FUNCTION_BLOCK Model (* Composite Function Block Type *)
  (* Standard: 61499-2 *)
  (* Version 0.0, 6/17/2016, Andrei, nxtControl GmbH, template *)
  PACKAGE Main;
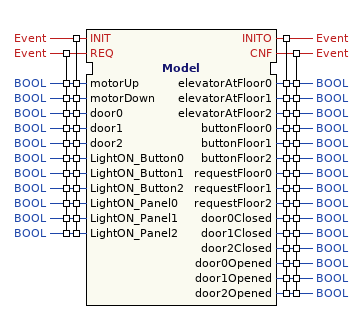
  EVENT_INPUT
    INIT WITH motorUp, motorDown, door0, door1, door2, LightON_Button0, LightON_Button1, LightON_Button2, LightON_Panel0, LightON_Panel1, LightON_Panel2; (* Initialization Request *)
    REQ WITH motorUp, motorDown, door0, door1, door2, LightON_Button0, LightON_Button1, LightON_Button2, LightON_Panel0, LightON_Panel1, LightON_Panel2; (* Normal Execution Request *)
  END_EVENT
  EVENT_OUTPUT
    INITO WITH buttonFloor0, buttonFloor1, buttonFloor2, requestFloor0, requestFloor1, requestFloor2, elevatorAtFloor0, elevatorAtFloor1, elevatorAtFloor2, door0Closed, door1Closed, door2Closed, door0Opened, door1Opened, door2Opened; (* Initialization Confirm *)
    CNF WITH buttonFloor0, buttonFloor1, buttonFloor2, requestFloor0, requestFloor1, requestFloor2, elevatorAtFloor0, elevatorAtFloor1, elevatorAtFloor2, door0Closed, door1Closed, door2Closed, door0Opened, door1Opened, door2Opened; (* Execution Confirmation *)
  END_EVENT
  VAR_INPUT
    motorUp : BOOL; (* Input event qualifier *)
    motorDown : BOOL;
    door0 : BOOL;
    door1 : BOOL;
    door2 : BOOL;
    LightON_Button0 : BOOL;
    LightON_Button1 : BOOL;
    LightON_Button2 : BOOL;
    LightON_Panel0 : BOOL;
    LightON_Panel1 : BOOL;
    LightON_Panel2 : BOOL;
  END_VAR
  VAR_OUTPUT
    elevatorAtFloor0 : BOOL;
    elevatorAtFloor1 : BOOL;
    elevatorAtFloor2 : BOOL;
    buttonFloor0 : BOOL; (* Output event qualifier *)
    buttonFloor1 : BOOL;
    buttonFloor2 : BOOL;
    requestFloor0 : BOOL;
    requestFloor1 : BOOL;
    requestFloor2 : BOOL;
    door0Closed : BOOL;
    door1Closed : BOOL;
    door2Closed : BOOL;
    door0Opened : BOOL;
    door1Opened : BOOL;
    door2Opened : BOOL;
  END_VAR
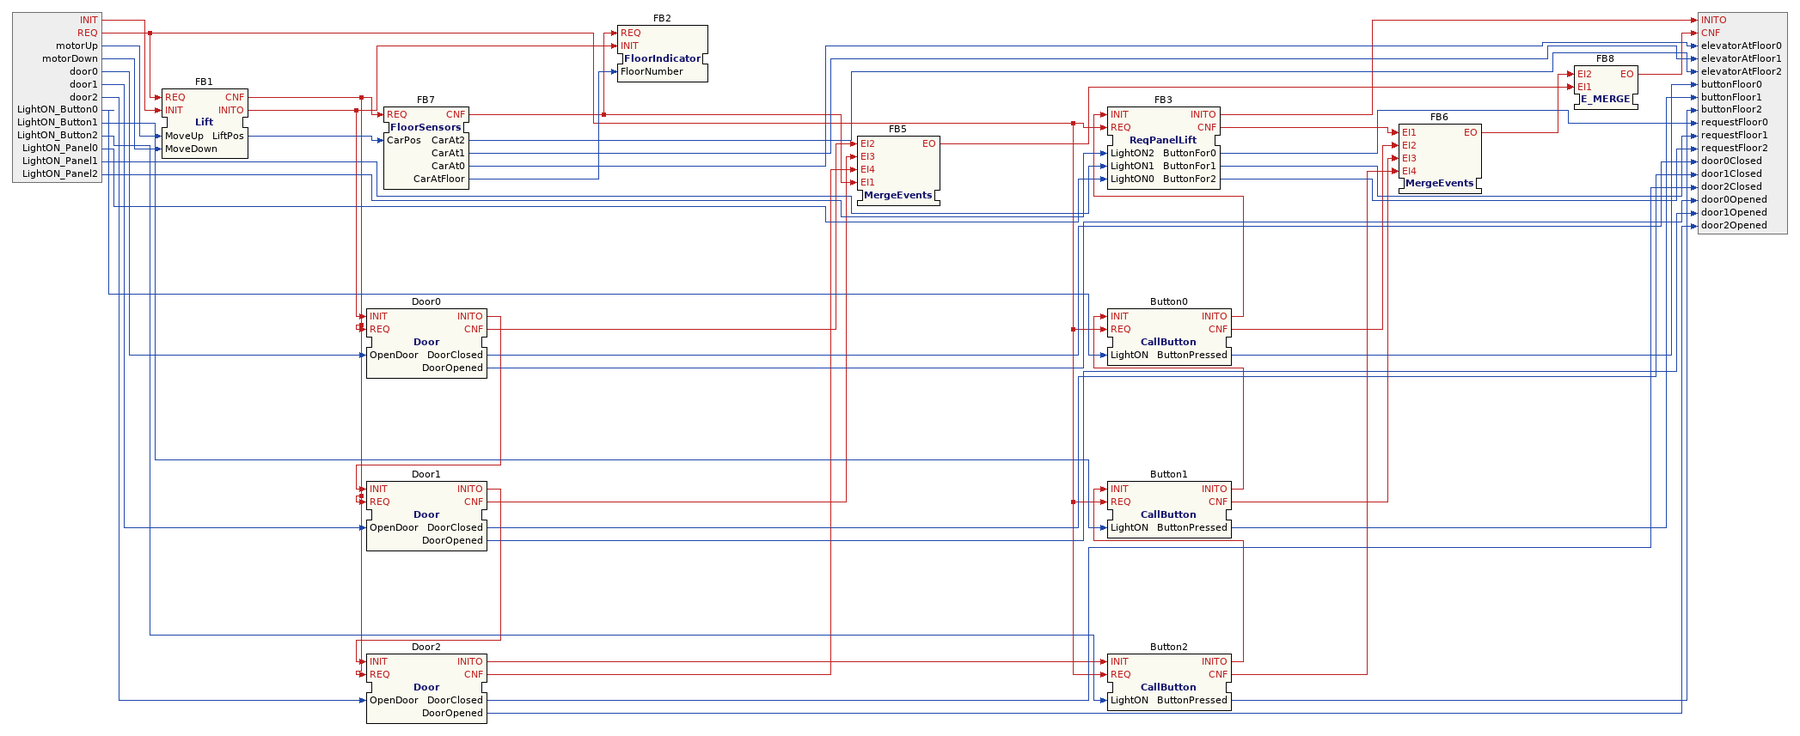
  FBS
    FB1 : Lift;
    FB2 : FloorIndicator;
    FB3 : ReqPanelLift;
    FB8 : E_MERGE;
    Door0 : Door;
    Door1 : Door;
    Door2 : Door;
    Button0 : CallButton;
    Button1 : CallButton;
    Button2 : CallButton;
    FB5 : MergeEvents;
    FB6 : MergeEvents;
    FB7 : FloorSensors;
  END_FBS
  EVENT_CONNECTIONS
    REQ TO FB1.REQ;
    INIT TO FB1.INIT;
    FB1.CNF TO FB7.REQ;
    FB1.INITO TO Door0.INIT;
    Door0.INITO TO Door1.INIT;
    Door1.INITO TO Door2.INIT;
    Door2.INITO TO Button2.INIT;
    Button2.INITO TO Button1.INIT;
    Button1.INITO TO Button0.INIT;
    Button0.INITO TO FB3.INIT;
    FB3.INITO TO INITO;
    FB7.CNF TO FB2.REQ;
    FB1.INITO TO FB2.INIT;
    FB8.EO TO CNF;
    Door0.CNF TO FB5.EI2;
    Door1.CNF TO FB5.EI3;
    Door2.CNF TO FB5.EI4;
    FB3.CNF TO FB6.EI1;
    Button0.CNF TO FB6.EI2;
    Button1.CNF TO FB6.EI3;
    Button2.CNF TO FB6.EI4;
    FB6.EO TO FB8.EI2;
    FB5.EO TO FB8.EI1;
    FB1.CNF TO Door1.REQ;
    FB1.CNF TO Door2.REQ;
    FB1.CNF TO Door0.REQ;
    REQ TO FB3.REQ;
    REQ TO Button0.REQ;
    REQ TO Button1.REQ;
    REQ TO Button2.REQ;
    FB7.CNF TO FB5.EI1;
  END_CONNECTIONS
  DATA_CONNECTIONS
    motorUp TO FB1.MoveUp;
    motorDown TO FB1.MoveDown;
    FB3.ButtonFor0 TO requestFloor0;
    FB3.ButtonFor1 TO requestFloor1;
    FB3.ButtonFor2 TO requestFloor2;
    FB1.LiftPos TO FB7.CarPos;
    FB7.CarAt2 TO elevatorAtFloor2;
    FB7.CarAt1 TO elevatorAtFloor1;
    FB7.CarAt0 TO elevatorAtFloor0;
    Door0.DoorClosed TO door0Closed;
    door0 TO Door0.OpenDoor;
    door1 TO Door1.OpenDoor;
    door2 TO Door2.OpenDoor;
    Door1.DoorClosed TO door1Closed;
    Door2.DoorClosed TO door2Closed;
    Button0.ButtonPressed TO buttonFloor0;
    Button1.ButtonPressed TO buttonFloor1;
    Button2.ButtonPressed TO buttonFloor2;
    FB7.CarAtFloor TO FB2.FloorNumber;
    Door2.DoorOpened TO door2Opened;
    Door1.DoorOpened TO door1Opened;
    Door0.DoorOpened TO door0Opened;
    LightON_Button2 TO Button2.LightON;
    LightON_Button1 TO Button1.LightON;
    LightON_Button0 TO Button0.LightON;
    LightON_Panel2 TO FB3.LightON2;
    LightON_Panel1 TO FB3.LightON1;
    LightON_Panel0 TO FB3.LightON0;
  END_CONNECTIONS
END_FUNCTION_BLOCK
